{attribute 'qualified_only'}
VAR_GLOBAL
	Input_State AT %I*: UINT;
	Output_State AT %Q*: UINT;
	ConnState AT %I*: UDINT;
	ConnCtrl AT %Q*: UDINT;
	Input_100 AT %I*: ARRAY[0..100] OF BYTE;
	Output_100 AT %Q*: ARRAY[0..100] OF BYTE;
END_VAR

(* stored: Version 1.1.0.1, ProductVersion 3.1.4024.10
   GVL GVL: Id {2a2f395b-d7b9-4e51-8d6a-920baec2752b} *)
